// TIA Portal V21 export
FUNCTION_BLOCK "FB604"   // FB604, LAD
TITLE = FB604
{ S7_Optimized_Access := 'FALSE' }
AUTHOR : PRECISE
FAMILY : PRECISE
// CIP FILLING
// stored: AutoNumber false, SetENOAutomatically false
   VAR_INPUT
      CipSelected : Bool;
      CycleEnable : Bool;
      CycleRunning : Bool;
      SecPulse : Bool;
      AlwaysTrue : Bool;
      ActualQuantity : Real;
      ActualConductivity : Real;
      DrainWeight : Real;
      ActualRepetition : Int;
      ParaIn { ExternalAccessible := 'False'; ExternalVisible := 'False'; ExternalWritable := 'False'} : "FillingInputs";
   END_VAR
   VAR_OUTPUT
      Started : Bool;
      SWZDV : Bool;   // For Utility Selection: 0-SW
      PWZDV : Bool;   // For Utility Selection: 1-PW
      WFIZDV : Bool;   // For Utility Selection: 2-WFI
      RinsePump : Bool;
      ParaOut : "FillingOutputs";
      FillTimeMinPV : DInt;   // For Filling Method Slection: 1-Time
      FillTimeSecPV : DInt;   // For Filling Method Slection: 1-Time
      PulsingTimePV : Int;   // For Purging Selection: Yes
      RinseTimePV : Int;
      StepStatus : String[60];
      Print : "FillingPrint";
      Print_1 : "PulsingPrint";
   END_VAR
   VAR_IN_OUT
      Over : Bool;
      OverTemp : Bool;
      LineValvesTemp : Bool;
      ZDVTemp : Bool;
      PulsingValveTemp : Bool;
      ActualFillQuantity : Real;
      FillQuantityToleranceCalc : Real := 3.0;   // For Filling Method Slection: 0-Weight
      Temp1 : Int;
      Temp2 : Int;
      SampledConductivity : Real;
      ConductivitySuccess : Bool;
      RE1 : Bool;
      RE2 : Bool;
      RE3 : Bool;
      LineValves : Bool;
   END_VAR
   VAR
      ValveOnDelayPV : Int;
      ValveOffDelayPV : Int;
      FillTimer { S7_SetPoint := 'True'} : "FB101";
      "Pulsing/Rinsing" { S7_SetPoint := 'True'} : "FB102";
      StepDelay { S7_SetPoint := 'True'} : "FB110";
      ResetPrintValues { S7_SetPoint := 'True'} : TON_TIME;
   END_VAR
   // // ParaOut.Out.LineValvesSw : Common Valves for SW
   // // ParaOut.Out.LineValvesPw : Common Valves for PW
   // // ParaOut.Out.LineValvesWfi : Common Valves for WFI
   VAR_TEMP   // added for the SCL form of the ladder/FBD networks
      _w1 : Bool;
      _w2 : Bool;
      _w3 : Bool;
   END_VAR
BEGIN

REGION Network 1: Reset Print Status on Start
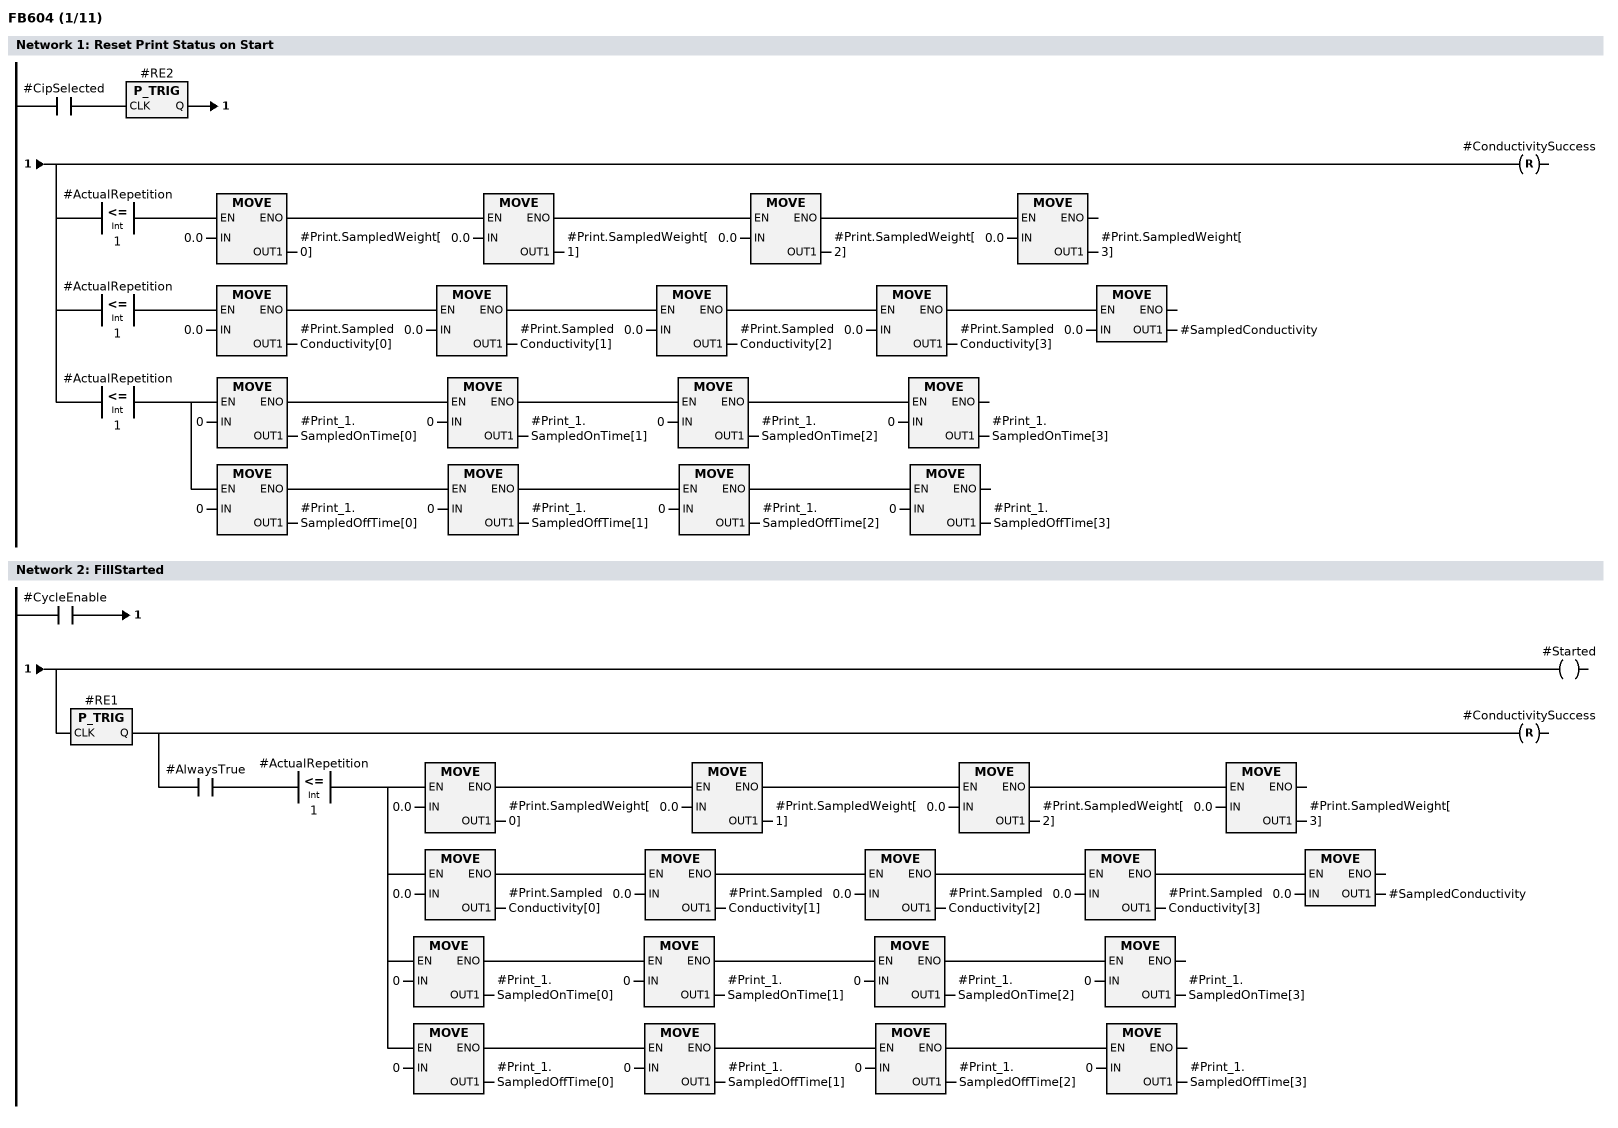
   RUNG wire#powerrail
      Contact( #CipSelected )
      P_Trig( #RE2 )
      wire#w1
      R_Coil( #ConductivitySuccess )
   END_RUNG
   RUNG wire#w1
      { S7_Templates := "SrcType := Int" } LE_Contact(in1 := #ActualRepetition, in2 := 1)
      Move(in := 0.0, out1 => #Print.SampledWeight[0])
      Move(in := 0.0, out1 => #Print.SampledWeight[1])
      Move(in := 0.0, out1 => #Print.SampledWeight[2])
      Move(in := 0.0, out1 => #Print.SampledWeight[3])
   END_RUNG
   RUNG wire#w1
      { S7_Templates := "SrcType := Int" } LE_Contact(in1 := #ActualRepetition, in2 := 1)
      Move(in := 0.0, out1 => #Print.SampledConductivity[0])
      Move(in := 0.0, out1 => #Print.SampledConductivity[1])
      Move(in := 0.0, out1 => #Print.SampledConductivity[2])
      Move(in := 0.0, out1 => #Print.SampledConductivity[3])
      Move(in := 0.0, out1 => #SampledConductivity)
   END_RUNG
   RUNG wire#w1
      { S7_Templates := "SrcType := Int" } LE_Contact(in1 := #ActualRepetition, in2 := 1)
      wire#w2
      Move(in := 0, out1 => #Print_1.SampledOnTime[0])
      Move(in := 0, out1 => #Print_1.SampledOnTime[1])
      Move(in := 0, out1 => #Print_1.SampledOnTime[2])
      Move(in := 0, out1 => #Print_1.SampledOnTime[3])
   END_RUNG
   RUNG wire#w2
      Move(in := 0, out1 => #Print_1.SampledOffTime[0])
      Move(in := 0, out1 => #Print_1.SampledOffTime[1])
      Move(in := 0, out1 => #Print_1.SampledOffTime[2])
      Move(in := 0, out1 => #Print_1.SampledOffTime[3])
   END_RUNG
   // the same network as SCL:
   #_w1 := #CipSelected AND NOT #RE2;   // rising edge
   #RE2 := #CipSelected;
   IF #_w1 THEN #ConductivitySuccess := FALSE; END_IF;
   IF #_w1 AND (#ActualRepetition <= 1) THEN
       #Print.SampledWeight[0] := 0.0;
       #Print.SampledWeight[1] := 0.0;
       #Print.SampledWeight[2] := 0.0;
       #Print.SampledWeight[3] := 0.0;
       #Print.SampledConductivity[0] := 0.0;
       #Print.SampledConductivity[1] := 0.0;
       #Print.SampledConductivity[2] := 0.0;
       #Print.SampledConductivity[3] := 0.0;
       #SampledConductivity := 0.0;
       #Print_1.SampledOnTime[0] := 0;
       #Print_1.SampledOnTime[1] := 0;
       #Print_1.SampledOnTime[2] := 0;
       #Print_1.SampledOnTime[3] := 0;
       #Print_1.SampledOffTime[0] := 0;
       #Print_1.SampledOffTime[1] := 0;
       #Print_1.SampledOffTime[2] := 0;
       #Print_1.SampledOffTime[3] := 0;
   END_IF;
END_REGION

REGION Network 2: FillStarted
   RUNG wire#powerrail
      Contact( #CycleEnable )
      wire#w1
      Coil( #Started )
   END_RUNG
   RUNG wire#w1
      P_Trig( #RE1 )
      wire#w2
      R_Coil( #ConductivitySuccess )
   END_RUNG
   RUNG wire#w2
      Contact( #AlwaysTrue )
      { S7_Templates := "SrcType := Int" } LE_Contact(in1 := #ActualRepetition, in2 := 1)
      wire#w3
      Move(in := 0.0, out1 => #Print.SampledWeight[0])
      Move(in := 0.0, out1 => #Print.SampledWeight[1])
      Move(in := 0.0, out1 => #Print.SampledWeight[2])
      Move(in := 0.0, out1 => #Print.SampledWeight[3])
   END_RUNG
   RUNG wire#w3
      Move(in := 0.0, out1 => #Print.SampledConductivity[0])
      Move(in := 0.0, out1 => #Print.SampledConductivity[1])
      Move(in := 0.0, out1 => #Print.SampledConductivity[2])
      Move(in := 0.0, out1 => #Print.SampledConductivity[3])
      Move(in := 0.0, out1 => #SampledConductivity)
   END_RUNG
   RUNG wire#w3
      Move(in := 0, out1 => #Print_1.SampledOnTime[0])
      Move(in := 0, out1 => #Print_1.SampledOnTime[1])
      Move(in := 0, out1 => #Print_1.SampledOnTime[2])
      Move(in := 0, out1 => #Print_1.SampledOnTime[3])
   END_RUNG
   RUNG wire#w3
      Move(in := 0, out1 => #Print_1.SampledOffTime[0])
      Move(in := 0, out1 => #Print_1.SampledOffTime[1])
      Move(in := 0, out1 => #Print_1.SampledOffTime[2])
      Move(in := 0, out1 => #Print_1.SampledOffTime[3])
   END_RUNG
   // the same network as SCL:
   #Started := #CycleEnable;
   #_w1 := #CycleEnable AND NOT #RE1;   // rising edge
   #RE1 := #CycleEnable;
   IF #_w1 THEN #ConductivitySuccess := FALSE; END_IF;
   IF #_w1 AND #AlwaysTrue AND (#ActualRepetition <= 1) THEN
       #Print.SampledWeight[0] := 0.0;
       #Print.SampledWeight[1] := 0.0;
       #Print.SampledWeight[2] := 0.0;
       #Print.SampledWeight[3] := 0.0;
       #Print.SampledConductivity[0] := 0.0;
       #Print.SampledConductivity[1] := 0.0;
       #Print.SampledConductivity[2] := 0.0;
       #Print.SampledConductivity[3] := 0.0;
       #SampledConductivity := 0.0;
       #Print_1.SampledOnTime[0] := 0;
       #Print_1.SampledOnTime[1] := 0;
       #Print_1.SampledOnTime[2] := 0;
       #Print_1.SampledOnTime[3] := 0;
       #Print_1.SampledOffTime[0] := 0;
       #Print_1.SampledOffTime[1] := 0;
       #Print_1.SampledOffTime[2] := 0;
       #Print_1.SampledOffTime[3] := 0;
   END_IF;
END_REGION

REGION Network 3: #InflightQuantity Calculation
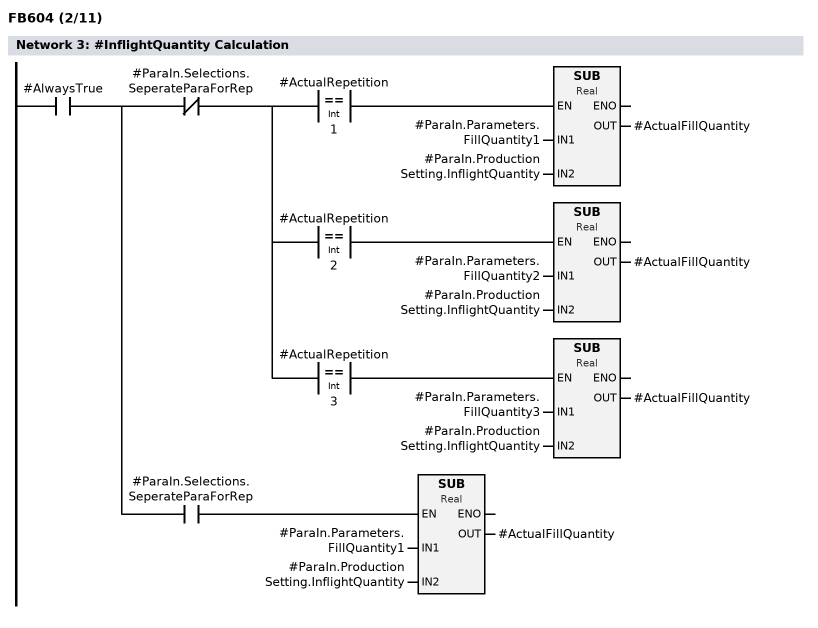
   RUNG wire#powerrail
      Contact( #AlwaysTrue )
      wire#w1
      I_Contact( #ParaIn.Selections.SeperateParaForRep )
      wire#w2
      { S7_Templates := "SrcType := Int" } EQ_Contact(in1 := #ActualRepetition, in2 := 1)
      { S7_Templates := "SrcType := Real"; S7_GenerateENO := "TRUE" } Sub(in1 := #ParaIn.Parameters.FillQuantity1, in2 := #ParaIn.ProductionSetting.InflightQuantity, out => #ActualFillQuantity)
   END_RUNG
   RUNG wire#w2
      { S7_Templates := "SrcType := Int" } EQ_Contact(in1 := #ActualRepetition, in2 := 2)
      { S7_Templates := "SrcType := Real"; S7_GenerateENO := "TRUE" } Sub(in1 := #ParaIn.Parameters.FillQuantity2, in2 := #ParaIn.ProductionSetting.InflightQuantity, out => #ActualFillQuantity)
   END_RUNG
   RUNG wire#w2
      { S7_Templates := "SrcType := Int" } EQ_Contact(in1 := #ActualRepetition, in2 := 3)
      { S7_Templates := "SrcType := Real"; S7_GenerateENO := "TRUE" } Sub(in1 := #ParaIn.Parameters.FillQuantity3, in2 := #ParaIn.ProductionSetting.InflightQuantity, out => #ActualFillQuantity)
   END_RUNG
   RUNG wire#w1
      Contact( #ParaIn.Selections.SeperateParaForRep )
      { S7_Templates := "SrcType := Real"; S7_GenerateENO := "TRUE" } Sub(in1 := #ParaIn.Parameters.FillQuantity1, in2 := #ParaIn.ProductionSetting.InflightQuantity, out => #ActualFillQuantity)
   END_RUNG
   // the same network as SCL:
   #_w1 := #AlwaysTrue AND NOT #ParaIn.Selections.SeperateParaForRep;
   IF #_w1 AND (#ActualRepetition = 1) THEN
       #ActualFillQuantity := #ParaIn.Parameters.FillQuantity1 - #ParaIn.ProductionSetting.InflightQuantity;
   END_IF;
   IF #_w1 AND (#ActualRepetition = 2) THEN
       #ActualFillQuantity := #ParaIn.Parameters.FillQuantity2 - #ParaIn.ProductionSetting.InflightQuantity;
   END_IF;
   IF #_w1 AND (#ActualRepetition = 3) THEN
       #ActualFillQuantity := #ParaIn.Parameters.FillQuantity3 - #ParaIn.ProductionSetting.InflightQuantity;
   END_IF;
   IF #AlwaysTrue AND #ParaIn.Selections.SeperateParaForRep THEN
       #ActualFillQuantity := #ParaIn.Parameters.FillQuantity1 - #ParaIn.ProductionSetting.InflightQuantity;
   END_IF;
END_REGION

REGION Network 4: Parameter for Time Based or Pulsing Method
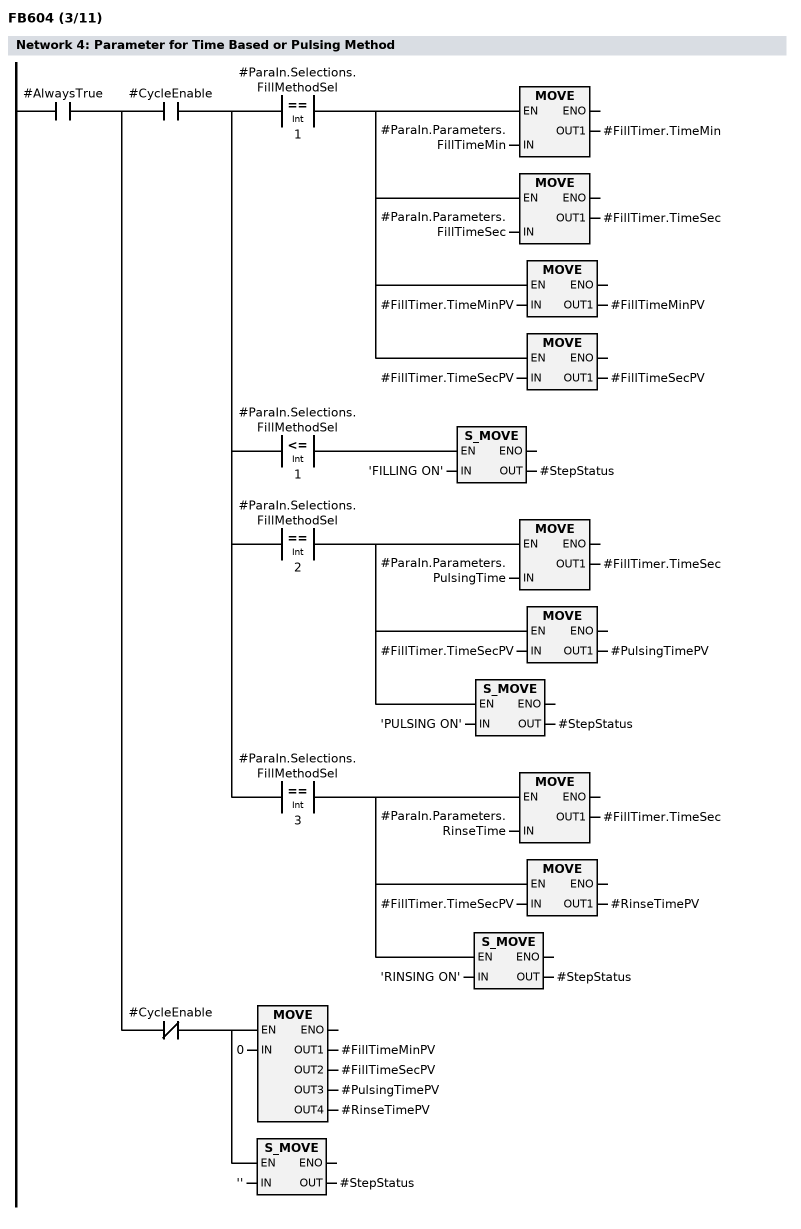
   RUNG wire#powerrail
      Contact( #AlwaysTrue )
      wire#w1
      Contact( #CycleEnable )
      wire#w2
      { S7_Templates := "SrcType := Int" } EQ_Contact(in1 := #ParaIn.Selections.FillMethodSel, in2 := 1)
      wire#w3
      Move(in := #ParaIn.Parameters.FillTimeMin, out1 => #FillTimer.TimeMin)
   END_RUNG
   RUNG wire#w3
      Move(in := #ParaIn.Parameters.FillTimeSec, out1 => #FillTimer.TimeSec)
   END_RUNG
   RUNG wire#w3
      Move(in := #FillTimer.TimeMinPV, out1 => #FillTimeMinPV)
   END_RUNG
   RUNG wire#w3
      Move(in := #FillTimer.TimeSecPV, out1 => #FillTimeSecPV)
   END_RUNG
   RUNG wire#w2
      { S7_Templates := "SrcType := Int" } LE_Contact(in1 := #ParaIn.Selections.FillMethodSel, in2 := 1)
      S_Move(in := 'FILLING ON', out => #StepStatus)
   END_RUNG
   RUNG wire#w2
      { S7_Templates := "SrcType := Int" } EQ_Contact(in1 := #ParaIn.Selections.FillMethodSel, in2 := 2)
      wire#w4
      Move(in := #ParaIn.Parameters.PulsingTime, out1 => #FillTimer.TimeSec)
   END_RUNG
   RUNG wire#w4
      Move(in := #FillTimer.TimeSecPV, out1 => #PulsingTimePV)
   END_RUNG
   RUNG wire#w4
      S_Move(in := 'PULSING ON', out => #StepStatus)
   END_RUNG
   RUNG wire#w2
      { S7_Templates := "SrcType := Int" } EQ_Contact(in1 := #ParaIn.Selections.FillMethodSel, in2 := 3)
      wire#w5
      Move(in := #ParaIn.Parameters.RinseTime, out1 => #FillTimer.TimeSec)
   END_RUNG
   RUNG wire#w5
      Move(in := #FillTimer.TimeSecPV, out1 => #RinseTimePV)
   END_RUNG
   RUNG wire#w5
      S_Move(in := 'RINSING ON', out => #StepStatus)
   END_RUNG
   RUNG wire#w1
      I_Contact( #CycleEnable )
      wire#w6
      Move(in := 0, out1 => #FillTimeMinPV, out2 => #FillTimeSecPV, out3 => #PulsingTimePV, out4 => #RinseTimePV)
   END_RUNG
   RUNG wire#w6
      S_Move(in := '', out => #StepStatus)
   END_RUNG
   // the same network as SCL:
   #_w1 := #AlwaysTrue AND #CycleEnable;
   IF #_w1 AND (#ParaIn.Selections.FillMethodSel = 1) THEN
       #FillTimer.TimeMin := #ParaIn.Parameters.FillTimeMin;
       #FillTimer.TimeSec := #ParaIn.Parameters.FillTimeSec;
       #FillTimeMinPV := #FillTimer.TimeMinPV;
       #FillTimeSecPV := #FillTimer.TimeSecPV;
   END_IF;
   IF #_w1 AND (#ParaIn.Selections.FillMethodSel <= 1) THEN #StepStatus := 'FILLING ON'; END_IF;
   IF #_w1 AND (#ParaIn.Selections.FillMethodSel = 2) THEN
       #FillTimer.TimeSec := #ParaIn.Parameters.PulsingTime;
       #PulsingTimePV := #FillTimer.TimeSecPV;
       #StepStatus := 'PULSING ON';
   END_IF;
   IF #_w1 AND (#ParaIn.Selections.FillMethodSel = 3) THEN
       #FillTimer.TimeSec := #ParaIn.Parameters.RinseTime;
       #RinseTimePV := #FillTimer.TimeSecPV;
       #StepStatus := 'RINSING ON';
   END_IF;
   IF #AlwaysTrue AND NOT #CycleEnable THEN
       #FillTimeMinPV := 0;
       #FillTimeSecPV := 0;
       #PulsingTimePV := 0;
       #RinseTimePV := 0;
       #StepStatus := '';
   END_IF;
END_REGION

REGION Network 5: Fill Timer / Pulsing Timer
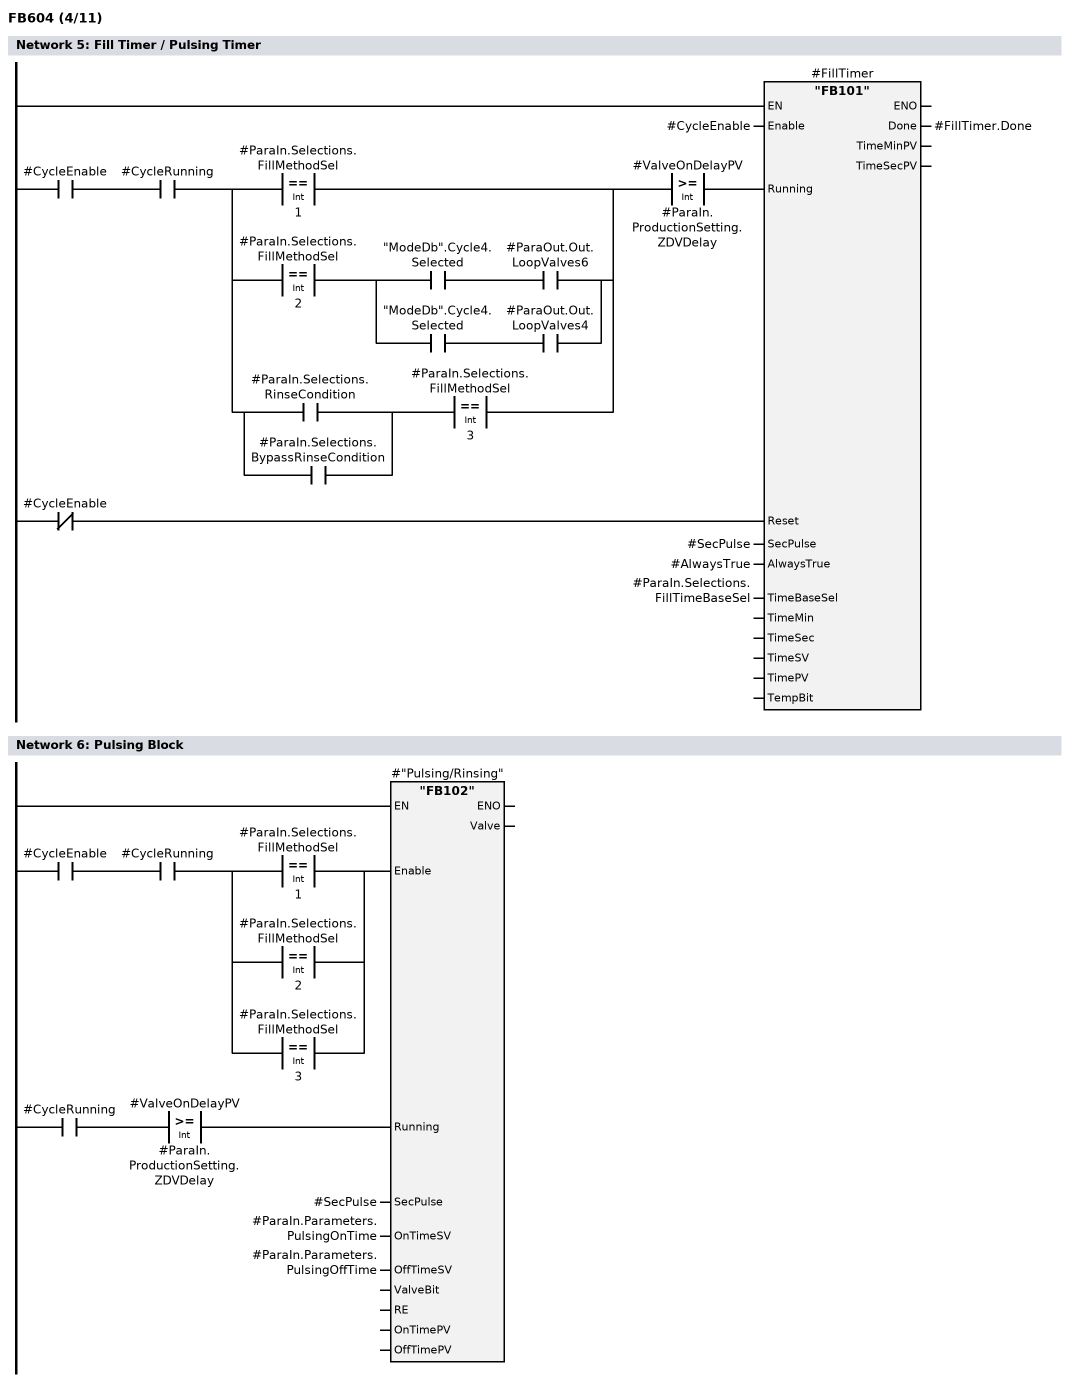
   RUNG wire#powerrail
      #FillTimer(Running := wire#w5, Reset := wire#w6, Enable := #CycleEnable, SecPulse := #SecPulse, AlwaysTrue := #AlwaysTrue, TimeBaseSel := #ParaIn.Selections.FillTimeBaseSel, TimeMin :=, TimeSec :=, TimeSV :=, TimePV :=, TempBit :=, Done => #FillTimer.Done, TimeMinPV =>, TimeSecPV =>)
   END_RUNG
   RUNG wire#powerrail
      Contact( #CycleEnable )
      Contact( #CycleRunning )
      wire#w1
      { S7_Templates := "SrcType := Int" } EQ_Contact(in1 := #ParaIn.Selections.FillMethodSel, in2 := 1)
      wire#w2
      { S7_Templates := "SrcType := Int" } GE_Contact(in1 := #ValveOnDelayPV, in2 := #ParaIn.ProductionSetting.ZDVDelay)
   END_RUNG wire#w5
   RUNG wire#w1
      { S7_Templates := "SrcType := Int" } EQ_Contact(in1 := #ParaIn.Selections.FillMethodSel, in2 := 2)
      wire#w3
      Contact( "ModeDb".Cycle4.Selected )
      Contact( #ParaOut.Out.LoopValves6 )
   END_RUNG wire#w2
   RUNG wire#w3
      Contact( "ModeDb".Cycle4.Selected )
      Contact( #ParaOut.Out.LoopValves4 )
   END_RUNG wire#w2
   RUNG wire#w1
      Contact( #ParaIn.Selections.RinseCondition )
      wire#w4
      { S7_Templates := "SrcType := Int" } EQ_Contact(in1 := #ParaIn.Selections.FillMethodSel, in2 := 3)
   END_RUNG wire#w2
   RUNG wire#w1
      Contact( #ParaIn.Selections.BypassRinseCondition )
   END_RUNG wire#w4
   RUNG wire#powerrail
      I_Contact( #CycleEnable )
   END_RUNG wire#w6
   // the same network as SCL:
   #FillTimer(Enable := #CycleEnable,   // "FB101"
              Running := #CycleEnable AND #CycleRunning AND ((#ParaIn.Selections.FillMethodSel = 1) OR ((#ParaIn.Selections.FillMethodSel = 2) AND (("ModeDb".Cycle4.Selected AND #ParaOut.Out.LoopValves6) OR ("ModeDb".Cycle4.Selected AND #ParaOut.Out.LoopValves4))) OR ((#ParaIn.Selections.RinseCondition OR #ParaIn.Selections.BypassRinseCondition) AND (#ParaIn.Selections.FillMethodSel = 3))) AND (#ValveOnDelayPV >= #ParaIn.ProductionSetting.ZDVDelay),
              Reset := NOT #CycleEnable,
              SecPulse := #SecPulse,
              AlwaysTrue := #AlwaysTrue,
              TimeBaseSel := #ParaIn.Selections.FillTimeBaseSel,
              Done => #FillTimer.Done);
END_REGION

REGION Network 6: Pulsing Block
   RUNG wire#powerrail
      #"Pulsing/Rinsing"(Enable := wire#w2, Running := wire#w3, SecPulse := #SecPulse, OnTimeSV := #ParaIn.Parameters.PulsingOnTime, OffTimeSV := #ParaIn.Parameters.PulsingOffTime, ValveBit :=, RE :=, OnTimePV :=, OffTimePV :=, Valve =>)
   END_RUNG
   RUNG wire#powerrail
      Contact( #CycleEnable )
      Contact( #CycleRunning )
      wire#w1
      { S7_Templates := "SrcType := Int" } EQ_Contact(in1 := #ParaIn.Selections.FillMethodSel, in2 := 1)
   END_RUNG wire#w2
   RUNG wire#w1
      { S7_Templates := "SrcType := Int" } EQ_Contact(in1 := #ParaIn.Selections.FillMethodSel, in2 := 2)
   END_RUNG wire#w2
   RUNG wire#w1
      { S7_Templates := "SrcType := Int" } EQ_Contact(in1 := #ParaIn.Selections.FillMethodSel, in2 := 3)
   END_RUNG wire#w2
   RUNG wire#powerrail
      Contact( #CycleRunning )
      { S7_Templates := "SrcType := Int" } GE_Contact(in1 := #ValveOnDelayPV, in2 := #ParaIn.ProductionSetting.ZDVDelay)
   END_RUNG wire#w3
   // the same network as SCL:
   #"Pulsing/Rinsing"(Enable := #CycleEnable AND #CycleRunning AND ((#ParaIn.Selections.FillMethodSel = 1) OR (#ParaIn.Selections.FillMethodSel = 2) OR (#ParaIn.Selections.FillMethodSel = 3)),   // "FB102"
                      Running := #CycleRunning AND (#ValveOnDelayPV >= #ParaIn.ProductionSetting.ZDVDelay),
                      SecPulse := #SecPulse,
                      OnTimeSV := #ParaIn.Parameters.PulsingOnTime,
                      OffTimeSV := #ParaIn.Parameters.PulsingOffTime);
END_REGION

REGION Network 7: Logic for Output
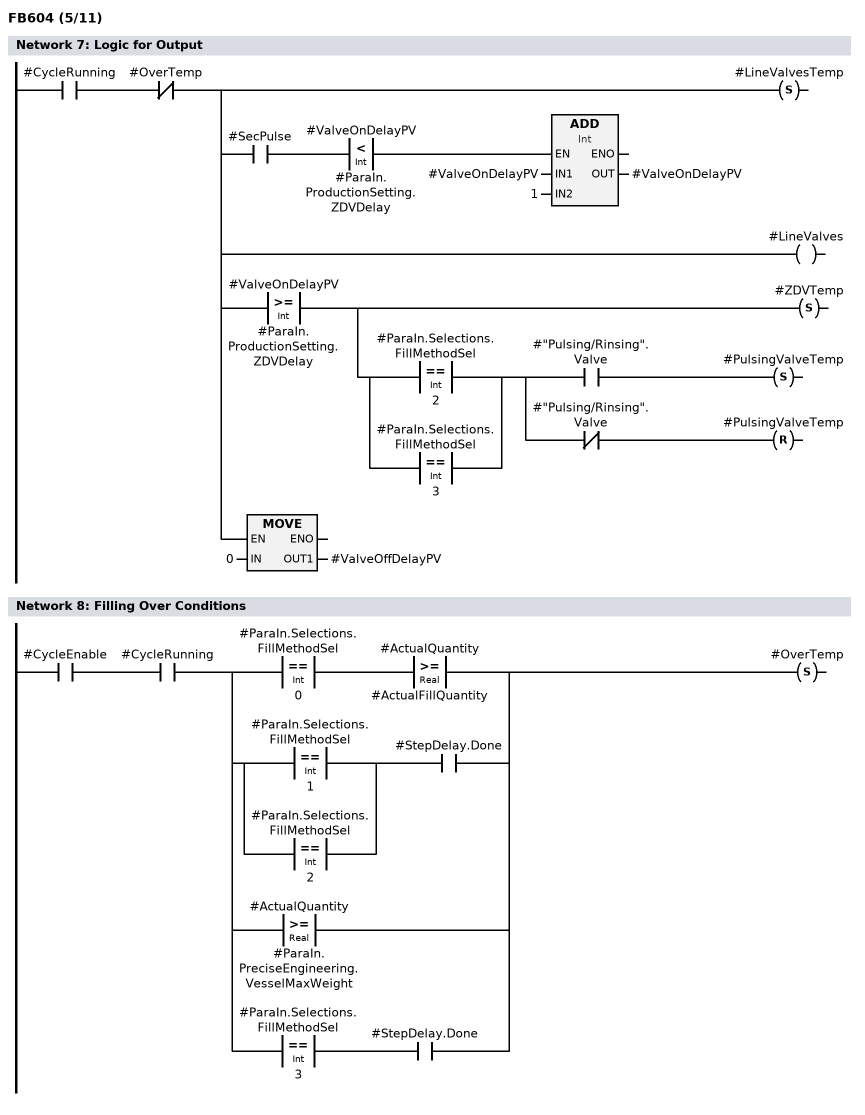
   RUNG wire#powerrail
      Contact( #CycleRunning )
      I_Contact( #OverTemp )
      wire#w1
      S_Coil( #LineValvesTemp )
   END_RUNG
   RUNG wire#w1
      Contact( #SecPulse )
      { S7_Templates := "SrcType := Int" } LT_Contact(in1 := #ValveOnDelayPV, in2 := #ParaIn.ProductionSetting.ZDVDelay)
      { S7_Templates := "SrcType := Int"; S7_GenerateENO := "TRUE" } Add(in1 := #ValveOnDelayPV, in2 := 1, out => #ValveOnDelayPV)
   END_RUNG
   RUNG wire#w1
      Coil( #LineValves )
   END_RUNG
   RUNG wire#w1
      { S7_Templates := "SrcType := Int" } GE_Contact(in1 := #ValveOnDelayPV, in2 := #ParaIn.ProductionSetting.ZDVDelay)
      wire#w2
      S_Coil( #ZDVTemp )
   END_RUNG
   RUNG wire#w2
      { S7_Templates := "SrcType := Int" } EQ_Contact(in1 := #ParaIn.Selections.FillMethodSel, in2 := 2)
      wire#w3
      Contact( #"Pulsing/Rinsing".Valve )
      S_Coil( #PulsingValveTemp )
   END_RUNG
   RUNG wire#w2
      { S7_Templates := "SrcType := Int" } EQ_Contact(in1 := #ParaIn.Selections.FillMethodSel, in2 := 3)
   END_RUNG wire#w3
   RUNG wire#w3
      I_Contact( #"Pulsing/Rinsing".Valve )
      R_Coil( #PulsingValveTemp )
   END_RUNG
   RUNG wire#w1
      { S7_GenerateENO := "TRUE" } Move(in := 0, out1 => #ValveOffDelayPV)
   END_RUNG
   // the same network as SCL:
   #_w1 := #CycleRunning AND NOT #OverTemp;
   IF #_w1 THEN #LineValvesTemp := TRUE; END_IF;
   IF #_w1 AND #SecPulse AND (#ValveOnDelayPV < #ParaIn.ProductionSetting.ZDVDelay) THEN
       #ValveOnDelayPV := #ValveOnDelayPV + 1;
   END_IF;
   #LineValves := #_w1;
   #_w2 := #_w1 AND (#ValveOnDelayPV >= #ParaIn.ProductionSetting.ZDVDelay);
   IF #_w2 THEN #ZDVTemp := TRUE; END_IF;
   #_w3 := #_w2 AND ((#ParaIn.Selections.FillMethodSel = 2) OR (#ParaIn.Selections.FillMethodSel = 3));
   IF #_w3 AND #"Pulsing/Rinsing".Valve THEN #PulsingValveTemp := TRUE; END_IF;
   IF #_w3 AND NOT #"Pulsing/Rinsing".Valve THEN #PulsingValveTemp := FALSE; END_IF;
   IF #_w1 THEN #ValveOffDelayPV := 0; END_IF;
END_REGION

REGION Network 8: Filling Over Conditions
   RUNG wire#powerrail
      Contact( #CycleEnable )
      Contact( #CycleRunning )
      wire#w1
      { S7_Templates := "SrcType := Int" } EQ_Contact(in1 := #ParaIn.Selections.FillMethodSel, in2 := 0)
      { S7_Templates := "SrcType := Real" } GE_Contact(in1 := #ActualQuantity, in2 := #ActualFillQuantity)
      wire#w2
      S_Coil( #OverTemp )
   END_RUNG
   RUNG wire#w1
      { S7_Templates := "SrcType := Int" } EQ_Contact(in1 := #ParaIn.Selections.FillMethodSel, in2 := 1)
      wire#w3
      Contact( #StepDelay.Done )
   END_RUNG wire#w2
   RUNG wire#w1
      { S7_Templates := "SrcType := Int" } EQ_Contact(in1 := #ParaIn.Selections.FillMethodSel, in2 := 2)
   END_RUNG wire#w3
   RUNG wire#w1
      { S7_Templates := "SrcType := Real" } GE_Contact(in1 := #ActualQuantity, in2 := #ParaIn.PreciseEngineering.VesselMaxWeight)
   END_RUNG wire#w2
   RUNG wire#w1
      { S7_Templates := "SrcType := Int" } EQ_Contact(in1 := #ParaIn.Selections.FillMethodSel, in2 := 3)
      Contact( #StepDelay.Done )
   END_RUNG wire#w2
   // the same network as SCL:
   IF #CycleEnable AND #CycleRunning AND (((#ParaIn.Selections.FillMethodSel = 0) AND (#ActualQuantity >= #ActualFillQuantity)) OR (((#ParaIn.Selections.FillMethodSel = 1) OR (#ParaIn.Selections.FillMethodSel = 2)) AND #StepDelay.Done) OR (#ActualQuantity >= #ParaIn.PreciseEngineering.VesselMaxWeight) OR ((#ParaIn.Selections.FillMethodSel = 3) AND #StepDelay.Done)) THEN
       #OverTemp := TRUE;
   END_IF;
END_REGION

REGION Network 9: Filling Done
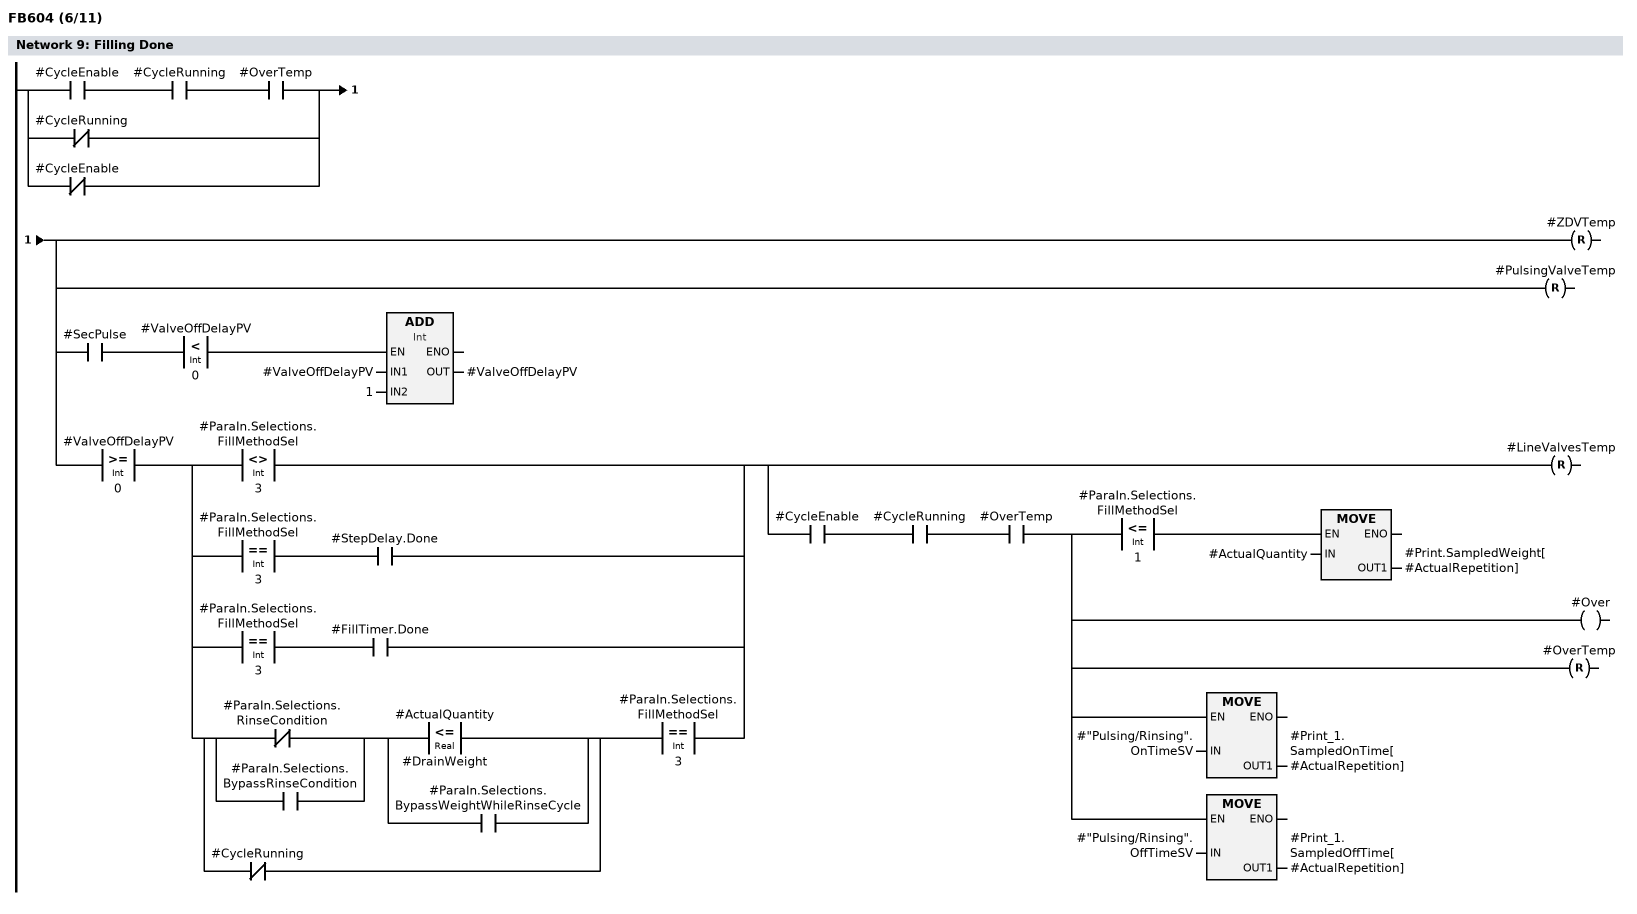
   RUNG wire#powerrail
      Contact( #CycleEnable )
      Contact( #CycleRunning )
      Contact( #OverTemp )
      wire#w1
      R_Coil( #ZDVTemp )
   END_RUNG
   RUNG wire#powerrail
      I_Contact( #CycleRunning )
   END_RUNG wire#w1
   RUNG wire#powerrail
      I_Contact( #CycleEnable )
   END_RUNG wire#w1
   RUNG wire#w1
      R_Coil( #PulsingValveTemp )
   END_RUNG
   RUNG wire#w1
      Contact( #SecPulse )
      { S7_Templates := "SrcType := Int" } LT_Contact(in1 := #ValveOffDelayPV, in2 := 0)
      { S7_Templates := "SrcType := Int"; S7_GenerateENO := "TRUE" } Add(in1 := #ValveOffDelayPV, in2 := 1, out => #ValveOffDelayPV)
   END_RUNG
   RUNG wire#w1
      { S7_Templates := "SrcType := Int" } GE_Contact(in1 := #ValveOffDelayPV, in2 := 0)
      wire#w2
      { S7_Templates := "SrcType := Int" } NE_Contact(in1 := #ParaIn.Selections.FillMethodSel, in2 := 3)
      wire#w3
      R_Coil( #LineValvesTemp )
   END_RUNG
   RUNG wire#w2
      { S7_Templates := "SrcType := Int" } EQ_Contact(in1 := #ParaIn.Selections.FillMethodSel, in2 := 3)
      Contact( #StepDelay.Done )
   END_RUNG wire#w3
   RUNG wire#w2
      { S7_Templates := "SrcType := Int" } EQ_Contact(in1 := #ParaIn.Selections.FillMethodSel, in2 := 3)
      Contact( #FillTimer.Done )
   END_RUNG wire#w3
   RUNG wire#w2
      I_Contact( #ParaIn.Selections.RinseCondition )
      wire#w4
      { S7_Templates := "SrcType := Real" } LE_Contact(in1 := #ActualQuantity, in2 := #DrainWeight)
      wire#w5
      { S7_Templates := "SrcType := Int" } EQ_Contact(in1 := #ParaIn.Selections.FillMethodSel, in2 := 3)
   END_RUNG wire#w3
   RUNG wire#w2
      Contact( #ParaIn.Selections.BypassRinseCondition )
   END_RUNG wire#w4
   RUNG wire#w4
      Contact( #ParaIn.Selections.BypassWeightWhileRinseCycle )
   END_RUNG wire#w5
   RUNG wire#w2
      I_Contact( #CycleRunning )
   END_RUNG wire#w5
   RUNG wire#w3
      Contact( #CycleEnable )
      Contact( #CycleRunning )
      Contact( #OverTemp )
      wire#w6
      { S7_Templates := "SrcType := Int" } LE_Contact(in1 := #ParaIn.Selections.FillMethodSel, in2 := 1)
      Move(in := #ActualQuantity, out1 => #Print.SampledWeight[#ActualRepetition])
   END_RUNG
   RUNG wire#w6
      Coil( #Over )
   END_RUNG
   RUNG wire#w6
      R_Coil( #OverTemp )
   END_RUNG
   RUNG wire#w6
      Move(in := #"Pulsing/Rinsing".OnTimeSV, out1 => #Print_1.SampledOnTime[#ActualRepetition])
   END_RUNG
   RUNG wire#w6
      Move(in := #"Pulsing/Rinsing".OffTimeSV, out1 => #Print_1.SampledOffTime[#ActualRepetition])
   END_RUNG
   // the same network as SCL:
   #_w1 := (#CycleEnable AND #CycleRunning AND #OverTemp) OR NOT #CycleRunning OR NOT #CycleEnable;
   IF #_w1 THEN
       #ZDVTemp := FALSE;
       #PulsingValveTemp := FALSE;
   END_IF;
   IF #_w1 AND #SecPulse AND (#ValveOffDelayPV < 0) THEN #ValveOffDelayPV := #ValveOffDelayPV + 1; END_IF;
   #_w2 := #_w1 AND (#ValveOffDelayPV >= 0) AND ((#ParaIn.Selections.FillMethodSel <> 3) OR ((#ParaIn.Selections.FillMethodSel = 3) AND #StepDelay.Done) OR ((#ParaIn.Selections.FillMethodSel = 3) AND #FillTimer.Done) OR ((((NOT #ParaIn.Selections.RinseCondition OR #ParaIn.Selections.BypassRinseCondition) AND ((#ActualQuantity <= #DrainWeight) OR #ParaIn.Selections.BypassWeightWhileRinseCycle)) OR NOT #CycleRunning) AND (#ParaIn.Selections.FillMethodSel = 3)));
   IF #_w2 THEN #LineValvesTemp := FALSE; END_IF;
   #_w3 := #_w2 AND #CycleEnable AND #CycleRunning AND #OverTemp;
   IF #_w3 AND (#ParaIn.Selections.FillMethodSel <= 1) THEN
       #Print.SampledWeight[#ActualRepetition] := #ActualQuantity;
   END_IF;
   #Over := #_w3;
   IF #_w3 THEN
       #OverTemp := FALSE;
       #Print_1.SampledOnTime[#ActualRepetition] := #"Pulsing/Rinsing".OnTimeSV;
       #Print_1.SampledOffTime[#ActualRepetition] := #"Pulsing/Rinsing".OffTimeSV;
   END_IF;
END_REGION

REGION Network 10: Output ON
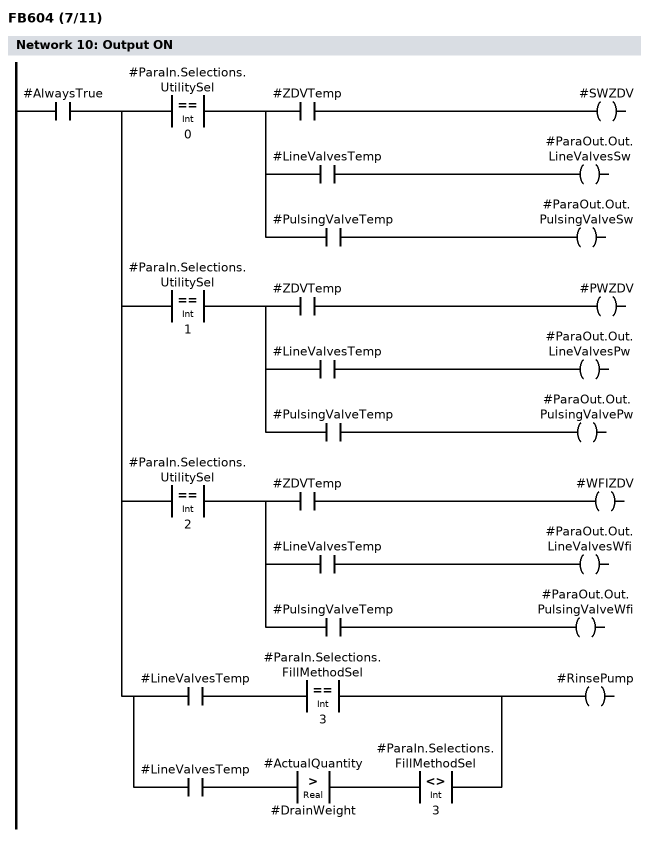
   RUNG wire#powerrail
      Contact( #AlwaysTrue )
      wire#w1
      { S7_Templates := "SrcType := Int" } EQ_Contact(in1 := #ParaIn.Selections.UtilitySel, in2 := 0)
      wire#w2
      Contact( #ZDVTemp )
      Coil( #SWZDV )
   END_RUNG
   RUNG wire#w2
      Contact( #LineValvesTemp )
      Coil( #ParaOut.Out.LineValvesSw )
   END_RUNG
   RUNG wire#w2
      Contact( #PulsingValveTemp )
      Coil( #ParaOut.Out.PulsingValveSw )
   END_RUNG
   RUNG wire#w1
      { S7_Templates := "SrcType := Int" } EQ_Contact(in1 := #ParaIn.Selections.UtilitySel, in2 := 1)
      wire#w3
      Contact( #ZDVTemp )
      Coil( #PWZDV )
   END_RUNG
   RUNG wire#w3
      Contact( #LineValvesTemp )
      Coil( #ParaOut.Out.LineValvesPw )
   END_RUNG
   RUNG wire#w3
      Contact( #PulsingValveTemp )
      Coil( #ParaOut.Out.PulsingValvePw )
   END_RUNG
   RUNG wire#w1
      { S7_Templates := "SrcType := Int" } EQ_Contact(in1 := #ParaIn.Selections.UtilitySel, in2 := 2)
      wire#w4
      Contact( #ZDVTemp )
      Coil( #WFIZDV )
   END_RUNG
   RUNG wire#w4
      Contact( #LineValvesTemp )
      Coil( #ParaOut.Out.LineValvesWfi )
   END_RUNG
   RUNG wire#w4
      Contact( #PulsingValveTemp )
      Coil( #ParaOut.Out.PulsingValveWfi )
   END_RUNG
   RUNG wire#w1
      Contact( #LineValvesTemp )
      { S7_Templates := "SrcType := Int" } EQ_Contact(in1 := #ParaIn.Selections.FillMethodSel, in2 := 3)
      wire#w5
      Coil( #RinsePump )
   END_RUNG
   RUNG wire#w1
      Contact( #LineValvesTemp )
      { S7_Templates := "SrcType := Real" } GT_Contact(in1 := #ActualQuantity, in2 := #DrainWeight)
      { S7_Templates := "SrcType := Int" } NE_Contact(in1 := #ParaIn.Selections.FillMethodSel, in2 := 3)
   END_RUNG wire#w5
   // the same network as SCL:
   #_w1 := #AlwaysTrue AND (#ParaIn.Selections.UtilitySel = 0);
   #SWZDV := #_w1 AND #ZDVTemp;
   #ParaOut.Out.LineValvesSw := #_w1 AND #LineValvesTemp;
   #ParaOut.Out.PulsingValveSw := #_w1 AND #PulsingValveTemp;
   #_w2 := #AlwaysTrue AND (#ParaIn.Selections.UtilitySel = 1);
   #PWZDV := #_w2 AND #ZDVTemp;
   #ParaOut.Out.LineValvesPw := #_w2 AND #LineValvesTemp;
   #ParaOut.Out.PulsingValvePw := #_w2 AND #PulsingValveTemp;
   #_w3 := #AlwaysTrue AND (#ParaIn.Selections.UtilitySel = 2);
   #WFIZDV := #_w3 AND #ZDVTemp;
   #ParaOut.Out.LineValvesWfi := #_w3 AND #LineValvesTemp;
   #ParaOut.Out.PulsingValveWfi := #_w3 AND #PulsingValveTemp;
   #RinsePump := #AlwaysTrue AND ((#LineValvesTemp AND (#ParaIn.Selections.FillMethodSel = 3)) OR (#LineValvesTemp AND (#ActualQuantity > #DrainWeight) AND (#ParaIn.Selections.FillMethodSel <> 3)));
END_REGION

REGION Network 11: StepDelay.StepTimeSv
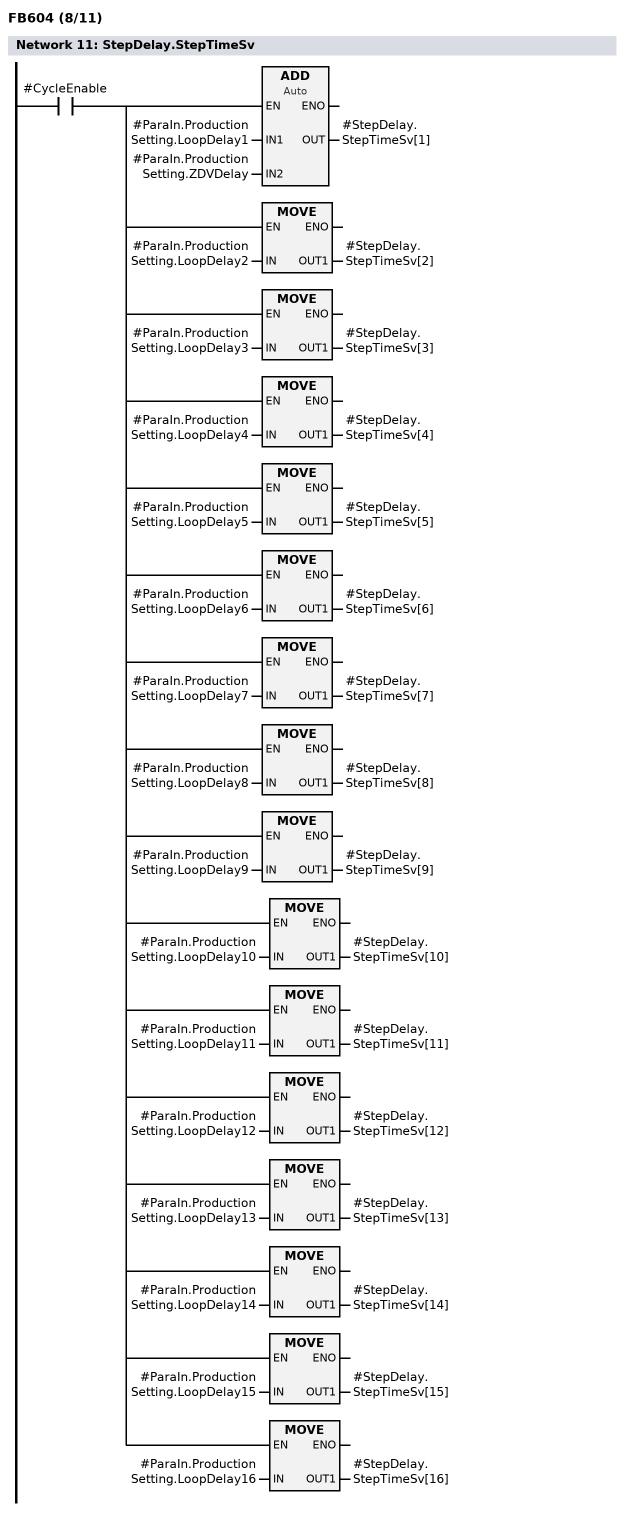
   RUNG wire#powerrail
      Contact( #CycleEnable )
      wire#w1
      Add(in1 := #ParaIn.ProductionSetting.LoopDelay1, in2 := #ParaIn.ProductionSetting.ZDVDelay, out => #StepDelay.StepTimeSv[1])
   END_RUNG
   RUNG wire#w1
      Move(in := #ParaIn.ProductionSetting.LoopDelay2, out1 => #StepDelay.StepTimeSv[2])
   END_RUNG
   RUNG wire#w1
      Move(in := #ParaIn.ProductionSetting.LoopDelay3, out1 => #StepDelay.StepTimeSv[3])
   END_RUNG
   RUNG wire#w1
      Move(in := #ParaIn.ProductionSetting.LoopDelay4, out1 => #StepDelay.StepTimeSv[4])
   END_RUNG
   RUNG wire#w1
      Move(in := #ParaIn.ProductionSetting.LoopDelay5, out1 => #StepDelay.StepTimeSv[5])
   END_RUNG
   RUNG wire#w1
      Move(in := #ParaIn.ProductionSetting.LoopDelay6, out1 => #StepDelay.StepTimeSv[6])
   END_RUNG
   RUNG wire#w1
      Move(in := #ParaIn.ProductionSetting.LoopDelay7, out1 => #StepDelay.StepTimeSv[7])
   END_RUNG
   RUNG wire#w1
      Move(in := #ParaIn.ProductionSetting.LoopDelay8, out1 => #StepDelay.StepTimeSv[8])
   END_RUNG
   RUNG wire#w1
      Move(in := #ParaIn.ProductionSetting.LoopDelay9, out1 => #StepDelay.StepTimeSv[9])
   END_RUNG
   RUNG wire#w1
      Move(in := #ParaIn.ProductionSetting.LoopDelay10, out1 => #StepDelay.StepTimeSv[10])
   END_RUNG
   RUNG wire#w1
      Move(in := #ParaIn.ProductionSetting.LoopDelay11, out1 => #StepDelay.StepTimeSv[11])
   END_RUNG
   RUNG wire#w1
      Move(in := #ParaIn.ProductionSetting.LoopDelay12, out1 => #StepDelay.StepTimeSv[12])
   END_RUNG
   RUNG wire#w1
      Move(in := #ParaIn.ProductionSetting.LoopDelay13, out1 => #StepDelay.StepTimeSv[13])
   END_RUNG
   RUNG wire#w1
      Move(in := #ParaIn.ProductionSetting.LoopDelay14, out1 => #StepDelay.StepTimeSv[14])
   END_RUNG
   RUNG wire#w1
      Move(in := #ParaIn.ProductionSetting.LoopDelay15, out1 => #StepDelay.StepTimeSv[15])
   END_RUNG
   RUNG wire#w1
      Move(in := #ParaIn.ProductionSetting.LoopDelay16, out1 => #StepDelay.StepTimeSv[16])
   END_RUNG
   // the same network as SCL:
   IF #CycleEnable THEN
       #StepDelay.StepTimeSv[1] := #ParaIn.ProductionSetting.LoopDelay1 + #ParaIn.ProductionSetting.ZDVDelay;
       #StepDelay.StepTimeSv[2] := #ParaIn.ProductionSetting.LoopDelay2;
       #StepDelay.StepTimeSv[3] := #ParaIn.ProductionSetting.LoopDelay3;
       #StepDelay.StepTimeSv[4] := #ParaIn.ProductionSetting.LoopDelay4;
       #StepDelay.StepTimeSv[5] := #ParaIn.ProductionSetting.LoopDelay5;
       #StepDelay.StepTimeSv[6] := #ParaIn.ProductionSetting.LoopDelay6;
       #StepDelay.StepTimeSv[7] := #ParaIn.ProductionSetting.LoopDelay7;
       #StepDelay.StepTimeSv[8] := #ParaIn.ProductionSetting.LoopDelay8;
       #StepDelay.StepTimeSv[9] := #ParaIn.ProductionSetting.LoopDelay9;
       #StepDelay.StepTimeSv[10] := #ParaIn.ProductionSetting.LoopDelay10;
       #StepDelay.StepTimeSv[11] := #ParaIn.ProductionSetting.LoopDelay11;
       #StepDelay.StepTimeSv[12] := #ParaIn.ProductionSetting.LoopDelay12;
       #StepDelay.StepTimeSv[13] := #ParaIn.ProductionSetting.LoopDelay13;
       #StepDelay.StepTimeSv[14] := #ParaIn.ProductionSetting.LoopDelay14;
       #StepDelay.StepTimeSv[15] := #ParaIn.ProductionSetting.LoopDelay15;
       #StepDelay.StepTimeSv[16] := #ParaIn.ProductionSetting.LoopDelay16;
   END_IF;
END_REGION

REGION Network 12: #StepDelay
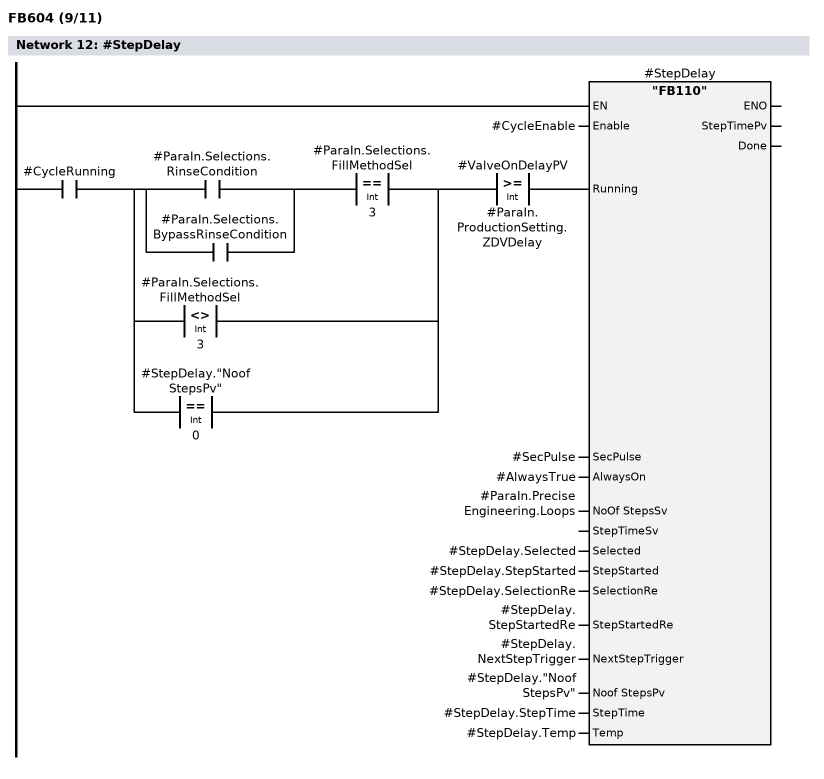
   RUNG wire#powerrail
      #StepDelay(Running := wire#w4, Enable := #CycleEnable, SecPulse := #SecPulse, AlwaysOn := #AlwaysTrue, "NoOf StepsSv" := #ParaIn.PreciseEngineering.Loops, StepTimeSv :=, Selected := #StepDelay.Selected, StepStarted := #StepDelay.StepStarted, SelectionRe := #StepDelay.SelectionRe, StepStartedRe := #StepDelay.StepStartedRe, NextStepTrigger := #StepDelay.NextStepTrigger, "Noof StepsPv" := #StepDelay."Noof StepsPv", StepTime := #StepDelay.StepTime, Temp := #StepDelay.Temp, StepTimePv =>, Done =>)
   END_RUNG
   RUNG wire#powerrail
      Contact( #CycleRunning )
      wire#w1
      Contact( #ParaIn.Selections.RinseCondition )
      wire#w2
      { S7_Templates := "SrcType := Int" } EQ_Contact(in1 := #ParaIn.Selections.FillMethodSel, in2 := 3)
      wire#w3
      { S7_Templates := "SrcType := Int" } GE_Contact(in1 := #ValveOnDelayPV, in2 := #ParaIn.ProductionSetting.ZDVDelay)
   END_RUNG wire#w4
   RUNG wire#w1
      Contact( #ParaIn.Selections.BypassRinseCondition )
   END_RUNG wire#w2
   RUNG wire#w1
      { S7_Templates := "SrcType := Int" } NE_Contact(in1 := #ParaIn.Selections.FillMethodSel, in2 := 3)
   END_RUNG wire#w3
   RUNG wire#w1
      { S7_Templates := "SrcType := Int" } EQ_Contact(in1 := #StepDelay."Noof StepsPv", in2 := 0)
   END_RUNG wire#w3
   // the same network as SCL:
   #StepDelay(Enable := #CycleEnable,   // "FB110"
              Running := #CycleRunning AND (((#ParaIn.Selections.RinseCondition OR #ParaIn.Selections.BypassRinseCondition) AND (#ParaIn.Selections.FillMethodSel = 3)) OR (#ParaIn.Selections.FillMethodSel <> 3) OR (#StepDelay."Noof StepsPv" = 0)) AND (#ValveOnDelayPV >= #ParaIn.ProductionSetting.ZDVDelay),
              SecPulse := #SecPulse,
              AlwaysOn := #AlwaysTrue,
              "NoOf StepsSv" := #ParaIn.PreciseEngineering.Loops,
              Selected := #StepDelay.Selected,
              StepStarted := #StepDelay.StepStarted,
              SelectionRe := #StepDelay.SelectionRe,
              StepStartedRe := #StepDelay.StepStartedRe,
              NextStepTrigger := #StepDelay.NextStepTrigger,
              "Noof StepsPv" := #StepDelay."Noof StepsPv",
              StepTime := #StepDelay.StepTime,
              Temp := #StepDelay.Temp);
END_REGION

REGION Network 13: Filling Loop Outputs
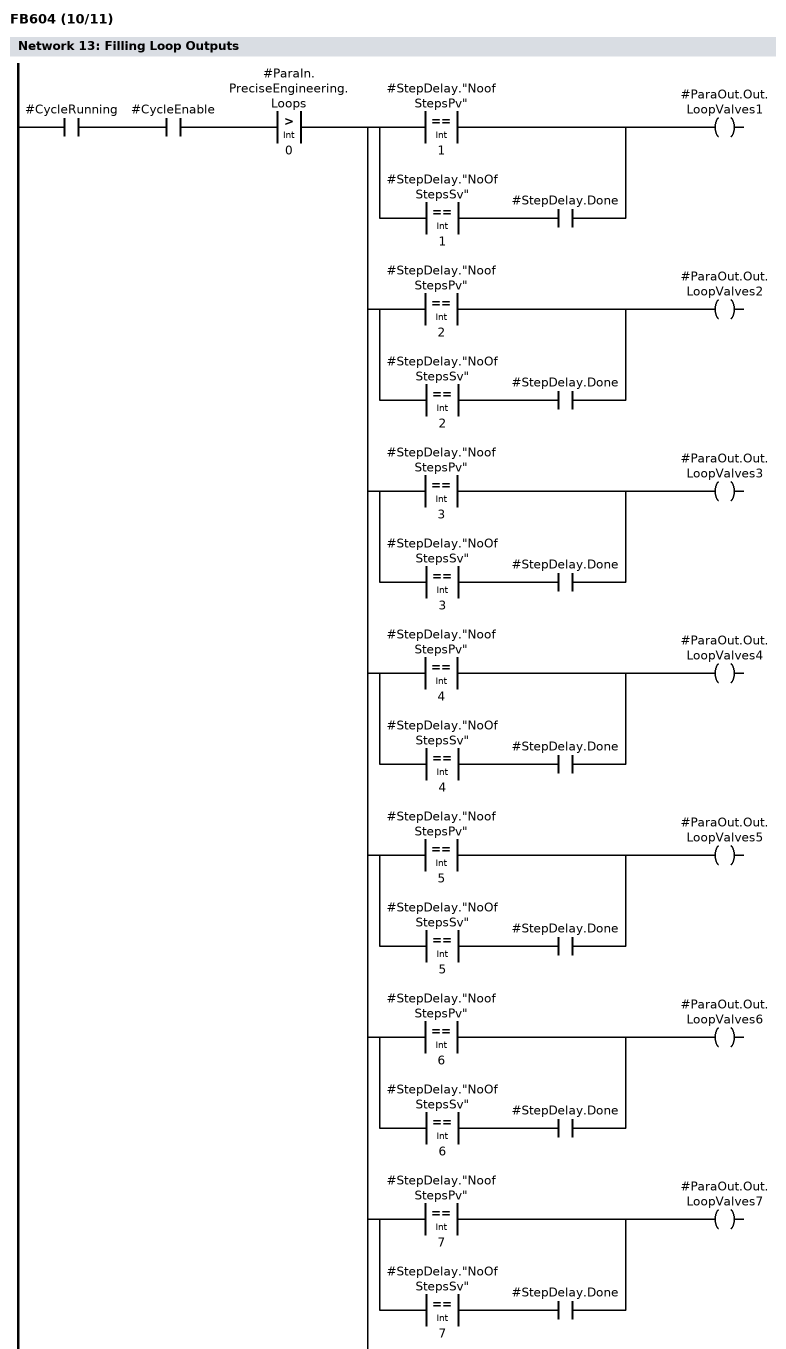
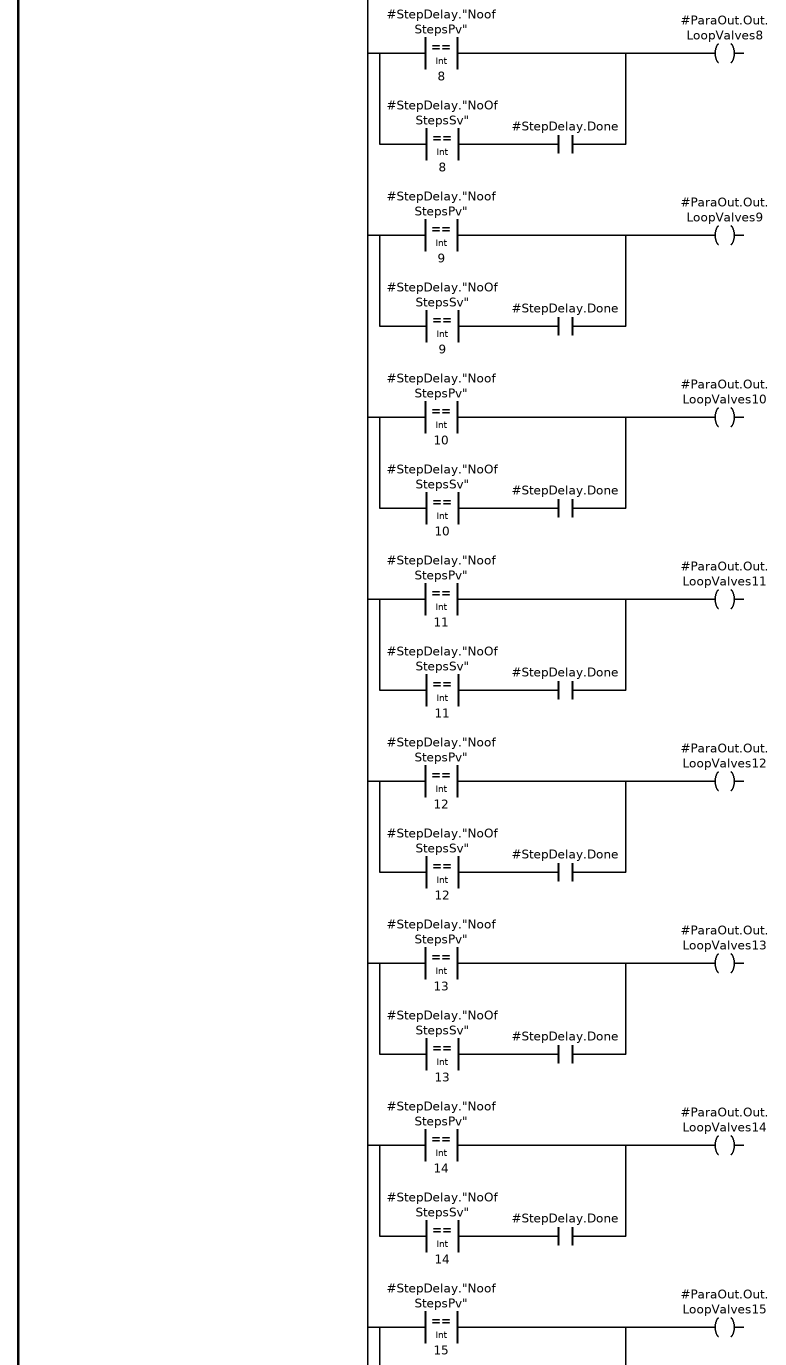
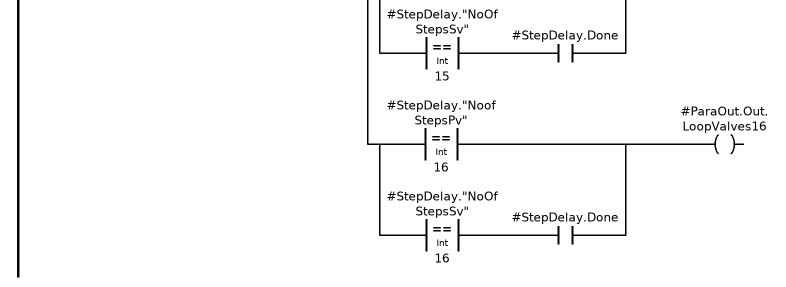
   RUNG wire#powerrail
      Contact( #CycleRunning )
      Contact( #CycleEnable )
      { S7_Templates := "SrcType := Int" } GT_Contact(in1 := #ParaIn.PreciseEngineering.Loops, in2 := 0)
      wire#w1
      { S7_Templates := "SrcType := Int" } EQ_Contact(in1 := #StepDelay."Noof StepsPv", in2 := 1)
      wire#w2
      Coil( #ParaOut.Out.LoopValves1 )
   END_RUNG
   RUNG wire#w1
      { S7_Templates := "SrcType := Int" } EQ_Contact(in1 := #StepDelay."NoOf StepsSv", in2 := 1)
      Contact( #StepDelay.Done )
   END_RUNG wire#w2
   RUNG wire#w1
      { S7_Templates := "SrcType := Int" } EQ_Contact(in1 := #StepDelay."Noof StepsPv", in2 := 2)
      wire#w3
      Coil( #ParaOut.Out.LoopValves2 )
   END_RUNG
   RUNG wire#w1
      { S7_Templates := "SrcType := Int" } EQ_Contact(in1 := #StepDelay."NoOf StepsSv", in2 := 2)
      Contact( #StepDelay.Done )
   END_RUNG wire#w3
   RUNG wire#w1
      { S7_Templates := "SrcType := Int" } EQ_Contact(in1 := #StepDelay."Noof StepsPv", in2 := 3)
      wire#w4
      Coil( #ParaOut.Out.LoopValves3 )
   END_RUNG
   RUNG wire#w1
      { S7_Templates := "SrcType := Int" } EQ_Contact(in1 := #StepDelay."NoOf StepsSv", in2 := 3)
      Contact( #StepDelay.Done )
   END_RUNG wire#w4
   RUNG wire#w1
      { S7_Templates := "SrcType := Int" } EQ_Contact(in1 := #StepDelay."Noof StepsPv", in2 := 4)
      wire#w5
      Coil( #ParaOut.Out.LoopValves4 )
   END_RUNG
   RUNG wire#w1
      { S7_Templates := "SrcType := Int" } EQ_Contact(in1 := #StepDelay."NoOf StepsSv", in2 := 4)
      Contact( #StepDelay.Done )
   END_RUNG wire#w5
   RUNG wire#w1
      { S7_Templates := "SrcType := Int" } EQ_Contact(in1 := #StepDelay."Noof StepsPv", in2 := 5)
      wire#w6
      Coil( #ParaOut.Out.LoopValves5 )
   END_RUNG
   RUNG wire#w1
      { S7_Templates := "SrcType := Int" } EQ_Contact(in1 := #StepDelay."NoOf StepsSv", in2 := 5)
      Contact( #StepDelay.Done )
   END_RUNG wire#w6
   RUNG wire#w1
      { S7_Templates := "SrcType := Int" } EQ_Contact(in1 := #StepDelay."Noof StepsPv", in2 := 6)
      wire#w7
      Coil( #ParaOut.Out.LoopValves6 )
   END_RUNG
   RUNG wire#w1
      { S7_Templates := "SrcType := Int" } EQ_Contact(in1 := #StepDelay."NoOf StepsSv", in2 := 6)
      Contact( #StepDelay.Done )
   END_RUNG wire#w7
   RUNG wire#w1
      { S7_Templates := "SrcType := Int" } EQ_Contact(in1 := #StepDelay."Noof StepsPv", in2 := 7)
      wire#w8
      Coil( #ParaOut.Out.LoopValves7 )
   END_RUNG
   RUNG wire#w1
      { S7_Templates := "SrcType := Int" } EQ_Contact(in1 := #StepDelay."NoOf StepsSv", in2 := 7)
      Contact( #StepDelay.Done )
   END_RUNG wire#w8
   RUNG wire#w1
      { S7_Templates := "SrcType := Int" } EQ_Contact(in1 := #StepDelay."Noof StepsPv", in2 := 8)
      wire#w9
      Coil( #ParaOut.Out.LoopValves8 )
   END_RUNG
   RUNG wire#w1
      { S7_Templates := "SrcType := Int" } EQ_Contact(in1 := #StepDelay."NoOf StepsSv", in2 := 8)
      Contact( #StepDelay.Done )
   END_RUNG wire#w9
   RUNG wire#w1
      { S7_Templates := "SrcType := Int" } EQ_Contact(in1 := #StepDelay."Noof StepsPv", in2 := 9)
      wire#w10
      Coil( #ParaOut.Out.LoopValves9 )
   END_RUNG
   RUNG wire#w1
      { S7_Templates := "SrcType := Int" } EQ_Contact(in1 := #StepDelay."NoOf StepsSv", in2 := 9)
      Contact( #StepDelay.Done )
   END_RUNG wire#w10
   RUNG wire#w1
      { S7_Templates := "SrcType := Int" } EQ_Contact(in1 := #StepDelay."Noof StepsPv", in2 := 10)
      wire#w11
      Coil( #ParaOut.Out.LoopValves10 )
   END_RUNG
   RUNG wire#w1
      { S7_Templates := "SrcType := Int" } EQ_Contact(in1 := #StepDelay."NoOf StepsSv", in2 := 10)
      Contact( #StepDelay.Done )
   END_RUNG wire#w11
   RUNG wire#w1
      { S7_Templates := "SrcType := Int" } EQ_Contact(in1 := #StepDelay."Noof StepsPv", in2 := 11)
      wire#w12
      Coil( #ParaOut.Out.LoopValves11 )
   END_RUNG
   RUNG wire#w1
      { S7_Templates := "SrcType := Int" } EQ_Contact(in1 := #StepDelay."NoOf StepsSv", in2 := 11)
      Contact( #StepDelay.Done )
   END_RUNG wire#w12
   RUNG wire#w1
      { S7_Templates := "SrcType := Int" } EQ_Contact(in1 := #StepDelay."Noof StepsPv", in2 := 12)
      wire#w13
      Coil( #ParaOut.Out.LoopValves12 )
   END_RUNG
   RUNG wire#w1
      { S7_Templates := "SrcType := Int" } EQ_Contact(in1 := #StepDelay."NoOf StepsSv", in2 := 12)
      Contact( #StepDelay.Done )
   END_RUNG wire#w13
   RUNG wire#w1
      { S7_Templates := "SrcType := Int" } EQ_Contact(in1 := #StepDelay."Noof StepsPv", in2 := 13)
      wire#w14
      Coil( #ParaOut.Out.LoopValves13 )
   END_RUNG
   RUNG wire#w1
      { S7_Templates := "SrcType := Int" } EQ_Contact(in1 := #StepDelay."NoOf StepsSv", in2 := 13)
      Contact( #StepDelay.Done )
   END_RUNG wire#w14
   RUNG wire#w1
      { S7_Templates := "SrcType := Int" } EQ_Contact(in1 := #StepDelay."Noof StepsPv", in2 := 14)
      wire#w15
      Coil( #ParaOut.Out.LoopValves14 )
   END_RUNG
   RUNG wire#w1
      { S7_Templates := "SrcType := Int" } EQ_Contact(in1 := #StepDelay."NoOf StepsSv", in2 := 14)
      Contact( #StepDelay.Done )
   END_RUNG wire#w15
   RUNG wire#w1
      { S7_Templates := "SrcType := Int" } EQ_Contact(in1 := #StepDelay."Noof StepsPv", in2 := 15)
      wire#w16
      Coil( #ParaOut.Out.LoopValves15 )
   END_RUNG
   RUNG wire#w1
      { S7_Templates := "SrcType := Int" } EQ_Contact(in1 := #StepDelay."NoOf StepsSv", in2 := 15)
      Contact( #StepDelay.Done )
   END_RUNG wire#w16
   RUNG wire#w1
      { S7_Templates := "SrcType := Int" } EQ_Contact(in1 := #StepDelay."Noof StepsPv", in2 := 16)
      wire#w17
      Coil( #ParaOut.Out.LoopValves16 )
   END_RUNG
   RUNG wire#w1
      { S7_Templates := "SrcType := Int" } EQ_Contact(in1 := #StepDelay."NoOf StepsSv", in2 := 16)
      Contact( #StepDelay.Done )
   END_RUNG wire#w17
   // the same network as SCL:
   #_w1 := #CycleRunning AND #CycleEnable AND (#ParaIn.PreciseEngineering.Loops > 0);
   #ParaOut.Out.LoopValves1 := #_w1 AND ((#StepDelay."Noof StepsPv" = 1) OR ((#StepDelay."NoOf StepsSv" = 1) AND #StepDelay.Done));
   #ParaOut.Out.LoopValves2 := #_w1 AND ((#StepDelay."Noof StepsPv" = 2) OR ((#StepDelay."NoOf StepsSv" = 2) AND #StepDelay.Done));
   #ParaOut.Out.LoopValves3 := #_w1 AND ((#StepDelay."Noof StepsPv" = 3) OR ((#StepDelay."NoOf StepsSv" = 3) AND #StepDelay.Done));
   #ParaOut.Out.LoopValves4 := #_w1 AND ((#StepDelay."Noof StepsPv" = 4) OR ((#StepDelay."NoOf StepsSv" = 4) AND #StepDelay.Done));
   #ParaOut.Out.LoopValves5 := #_w1 AND ((#StepDelay."Noof StepsPv" = 5) OR ((#StepDelay."NoOf StepsSv" = 5) AND #StepDelay.Done));
   #ParaOut.Out.LoopValves6 := #_w1 AND ((#StepDelay."Noof StepsPv" = 6) OR ((#StepDelay."NoOf StepsSv" = 6) AND #StepDelay.Done));
   #ParaOut.Out.LoopValves7 := #_w1 AND ((#StepDelay."Noof StepsPv" = 7) OR ((#StepDelay."NoOf StepsSv" = 7) AND #StepDelay.Done));
   #ParaOut.Out.LoopValves8 := #_w1 AND ((#StepDelay."Noof StepsPv" = 8) OR ((#StepDelay."NoOf StepsSv" = 8) AND #StepDelay.Done));
   #ParaOut.Out.LoopValves9 := #_w1 AND ((#StepDelay."Noof StepsPv" = 9) OR ((#StepDelay."NoOf StepsSv" = 9) AND #StepDelay.Done));
   #ParaOut.Out.LoopValves10 := #_w1 AND ((#StepDelay."Noof StepsPv" = 10) OR ((#StepDelay."NoOf StepsSv" = 10) AND #StepDelay.Done));
   #ParaOut.Out.LoopValves11 := #_w1 AND ((#StepDelay."Noof StepsPv" = 11) OR ((#StepDelay."NoOf StepsSv" = 11) AND #StepDelay.Done));
   #ParaOut.Out.LoopValves12 := #_w1 AND ((#StepDelay."Noof StepsPv" = 12) OR ((#StepDelay."NoOf StepsSv" = 12) AND #StepDelay.Done));
   #ParaOut.Out.LoopValves13 := #_w1 AND ((#StepDelay."Noof StepsPv" = 13) OR ((#StepDelay."NoOf StepsSv" = 13) AND #StepDelay.Done));
   #ParaOut.Out.LoopValves14 := #_w1 AND ((#StepDelay."Noof StepsPv" = 14) OR ((#StepDelay."NoOf StepsSv" = 14) AND #StepDelay.Done));
   #ParaOut.Out.LoopValves15 := #_w1 AND ((#StepDelay."Noof StepsPv" = 15) OR ((#StepDelay."NoOf StepsSv" = 15) AND #StepDelay.Done));
   #ParaOut.Out.LoopValves16 := #_w1 AND ((#StepDelay."Noof StepsPv" = 16) OR ((#StepDelay."NoOf StepsSv" = 16) AND #StepDelay.Done));
END_REGION

REGION Network 14: Reset
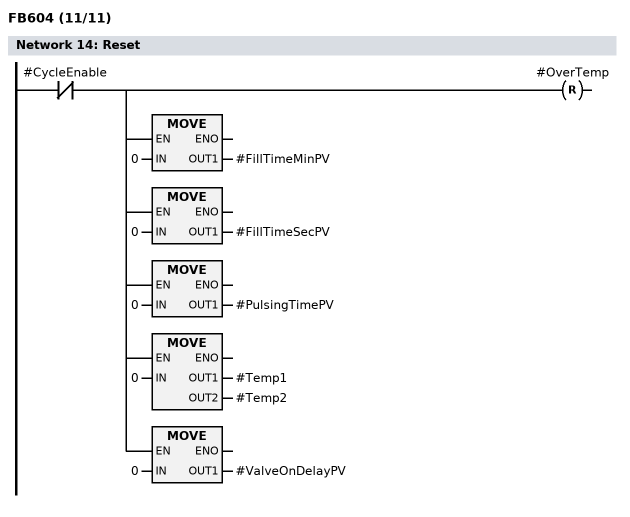
   RUNG wire#powerrail
      I_Contact( #CycleEnable )
      wire#w1
      R_Coil( #OverTemp )
   END_RUNG
   RUNG wire#w1
      { S7_GenerateENO := "TRUE" } Move(in := 0, out1 => #FillTimeMinPV)
   END_RUNG
   RUNG wire#w1
      { S7_GenerateENO := "TRUE" } Move(in := 0, out1 => #FillTimeSecPV)
   END_RUNG
   RUNG wire#w1
      { S7_GenerateENO := "TRUE" } Move(in := 0, out1 => #PulsingTimePV)
   END_RUNG
   RUNG wire#w1
      Move(in := 0, out1 => #Temp1, out2 => #Temp2)
   END_RUNG
   RUNG wire#w1
      { S7_GenerateENO := "TRUE" } Move(in := 0, out1 => #ValveOnDelayPV)
   END_RUNG
   // the same network as SCL:
   IF NOT #CycleEnable THEN
       #OverTemp := FALSE;
       #FillTimeMinPV := 0;
       #FillTimeSecPV := 0;
       #PulsingTimePV := 0;
       #Temp1 := 0;
       #Temp2 := 0;
       #ValveOnDelayPV := 0;
   END_IF;
END_REGION
END_FUNCTION_BLOCK
